RoboDK station: Welding_Cell.rdk

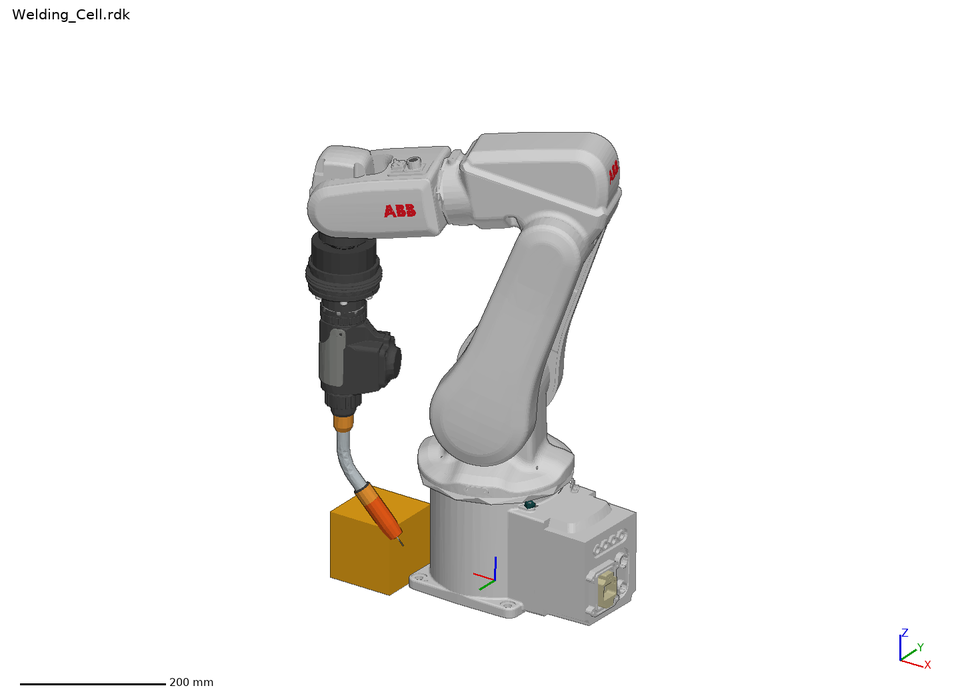
[picture v0: the station drawn from its stored meshes, robots at their saved joint values, targets as dots, program paths as lines]
Station Welding_Cell_v1 (saved by RoboDK 6.0.1). Poses are relative to the parent item; angles as X-Y-Z fixed-axis rotations.
  - frame ABB IRB 120-3/0.6 Base at (1189.63, 59.41, -0.41) mm, rotated rx 0.4 ry 0 rz 179.33 deg
    - robot ABB IRB 120-3/0.6: 6 axes, payload 3 kg, reach 580 mm, repeatability 0.01 mm, weight 25 kg
        modified DH rows (alpha deg, a mm, theta deg, d mm): 0, 0, 0, 290; -90, 0, -90, 0; 0, 270, 0, 0; -90, 70, 0, 302; 90, 0, 0, 0; -90, 0, 180, 72
        joint limits [-165, -110, -90, -160, -120, -400] to [165, 110, 70, 160, 120, 400]; home [0, 0, 0, 0, 0, 0]; saved at [21, -20, 30, 0, 80, 0]
      - tool Fronius MTB500i Welding Gun, TCP at (86, 0, 451.5) mm, rotated rx 0 ry 36 rz 0 deg, size 139 x 105 x 455.9 mm
  - object Cube 100mm at (952.65, 1.6, -38.25) mm, size 100 x 100 x 100 mm, geometry from Cube-100mm.sld
  - Python program Prog1 (listed below)

--- Python program Prog1 ---
from robodk.robolink import Robolink, ITEM_TYPE_ROBOT
import sys

RDK = Robolink()
robot_abb = RDK.Item('ABB IRB 120-3/0.6', ITEM_TYPE_ROBOT)

if not robot_abb.Valid():
    raise Exception("Nie znaleziono robota!")

RDK.setCollisionActive(1)
WELD_SPEED = 50
TRAVEL_SPEED = 150

weld_trajectory = [
    [ 21, -20, 30, 0, 80, 0],
    [ 10, -30, 30, 0, 80, 0],
    [  0, -30, 30, 0, 80, 0],
    [-10, -30, 30, 0, 80, 0],
    [-14, -30, 30, 0, 80, 0],
]

robot_abb.setSpeed(TRAVEL_SPEED)
robot_abb.MoveJ(robot_abb.JointsHome())

robot_abb.setSpeed(WELD_SPEED)
for joints in weld_trajectory:
    if RDK.Collisions() > 0:
        print("KOLIZJA!!! STOP")
        sys.exit()
    robot_abb.MoveJ(joints)

robot_abb.setSpeed(TRAVEL_SPEED)
robot_abb.MoveJ(robot_abb.JointsHome())
